(* IEC 61131-3 sources: POMIRTS_lab3/AS/Library/AsEPL, 3 files *)

(* ---- AsEPL.typ ---- *)
(********************************************************************
 * COPYRIGHT -- Bernecker + Rainer
 ********************************************************************
 * Library: AsEPL
 * File: AsEPL.typ
 * Author: B+R
 ********************************************************************
 * Data types of library AsEPL
 ********************************************************************)

TYPE
	EPL_I_TYPE : STRUCT			(*internal use*)
		init	: UDINT ;
		hdl	: UDINT ;
		st	: UDINT ;
		errInfo	: UDINT ;
		size	: UDINT ;
		bus	: USINT ;
		sl	: USINT ;
		ss	: USINT ;
		if_	: USINT ;
		nd	: USINT ;
		tid	: UDINT ;
	END_STRUCT;
END_TYPE

(* ---- AsEPL.fun ---- *)
(********************************************************************
 * COPYRIGHT -- Bernecker + Rainer
 ********************************************************************
 * Library: AsEPL
 * File: AsEPL.fun
 * Author: B+R
 ********************************************************************
 * Functions and function blocks of library AsEPL
 ********************************************************************)

FUNCTION_BLOCK EplSDORead					(*reads node's object entries when using an SDO transfer*)
	VAR_INPUT
		enable	:BOOL;						(*enables execution*)
		pDevice	:REFERENCE TO STRING[80];	(*device name given as a pointer, e.g., "SL<x>.SS<y>.IF<z>"*)
		node	:USINT;						(*address of the node to be read (1-127 or 0 for local OD)*)
		index	:UINT;						(*number of the index entry to be read*)
		subindex	:USINT;					(*number of the subindex entry to be read*)
		pData	:UDINT;						(*pointer to the buffer for read data*)
		datalen	:UDINT;						(*maximum length of the data to be read*)
	END_VAR

	VAR_OUTPUT
		status	:UINT;						(*execution status: ERR_OK, ERR_FUB_ENABLE_FALSE, 0xXXXX = see help*)
		errorinfo	:UDINT;					(*SDO Abort Code, e.g., EPL_ERR_SDO_PROTOCOL_TIMEOUT, EPL_ERR_SDO_COMMAND_ID_INVALID, ..*)
		readlen	:UDINT;						(*length of the entry read*)
	END_VAR

	VAR
		intern	:EPL_I_TYPE;				(*internal variable*)
	END_VAR
END_FUNCTION_BLOCK

FUNCTION_BLOCK EplSDOWrite					(*writes a node's object entries when using an SDO transfer*)
	VAR_INPUT
		enable	:BOOL;						(*enables execution*)
		pDevice	:REFERENCE TO STRING[80];	(*device name given as a pointer, e.g., "SL<x>.SS<y>.IF<z>"*)
		node	:USINT;						(*address of the node to be written (1-255 or 0 for local OD)*)
		index	:UINT;						(*number of the index entry to be written*)
		subindex	:USINT;					(*number of the subindex entry to be written*)
		pData	:UDINT;						(*pointer to the data to be written*)
		datalen	:UDINT;						(*length of the data to be written*)
	END_VAR

	VAR_OUTPUT
		status	:UINT;						(*execution status: ERR_OK, ERR_FUB_ENABLE_FALSE, 0xXXXX = see help*)
		errorinfo	:UDINT;					(*SDO abort code, e.g., EPL_ERR_SDO_PROTOCOL_TIMEOUT, EPL_ERR_SDO_COMMAND_ID_INVALID, ..*)
	END_VAR

	VAR
		intern	:EPL_I_TYPE;				(*internal variable*)
	END_VAR
END_FUNCTION_BLOCK

FUNCTION_BLOCK EplGetLocalNodeID			(*queries the local node address of the PLC*)
	VAR_INPUT
		enable	:BOOL;						(*enables execution*)
		pDevice	:REFERENCE TO STRING[80];	(*device name given as a pointer, e.g., "SL<x>.SS<y>.IF<z>"*)
	END_VAR

	VAR_OUTPUT
		status	:UINT;						(*execution status: ERR_OK, ERR_FUB_ENABLE_FALSE, 0xXXXX = see help*)
		nodeid	:USINT;						(*local node number of the PLC*)
	END_VAR
END_FUNCTION_BLOCK

(* ---- AsEPL.var ---- *)
(********************************************************************
 * COPYRIGHT -- Bernecker + Rainer
 ********************************************************************
 * Library: AsEPL
 * File: AsEPL.var
 * Author: B+R
 ********************************************************************
 * Local variables of library AsEPL
 ********************************************************************)

VAR CONSTANT
	ERR_ASEPL_NOT_IMPLEMENTED	: UINT	:= 31399;	(*error code for non-implemented functionality*)
	ERR_ASEPL_ACCESS_FAILED	: UINT	:= 31344;		(*read or write access failed*)
	ERR_ASEPL_WRONG_DEVICE	: UINT	:= 31341;		(*specified device not a POWERLINK interface*)
	ERR_ASEPL_MN_ONLY	: UINT	:= 31342;			(*function can only be executed on an MN (managing node)*)
	ERR_ASEPL_CN_ONLY	: UINT	:= 31343;			(*function can only be executed on a CN (controlled node)*)
	ERR_ASEPL_BASE	: UINT	:= 31340;				(*base error number*)
END_VAR
